FUNCTION_BLOCK LEDStateMachine
VAR_INPUT
END_VAR
VAR_OUTPUT
END_VAR
VAR
END_VAR

END_FUNCTION_BLOCK

(* stored: Version 1.1.0.1, ProductVersion 3.1.4024.12
   POU LEDStateMachine: Id {11a7e2b3-5e04-4b6a-9c94-27e77c703e44}, SpecialFunc None *)
